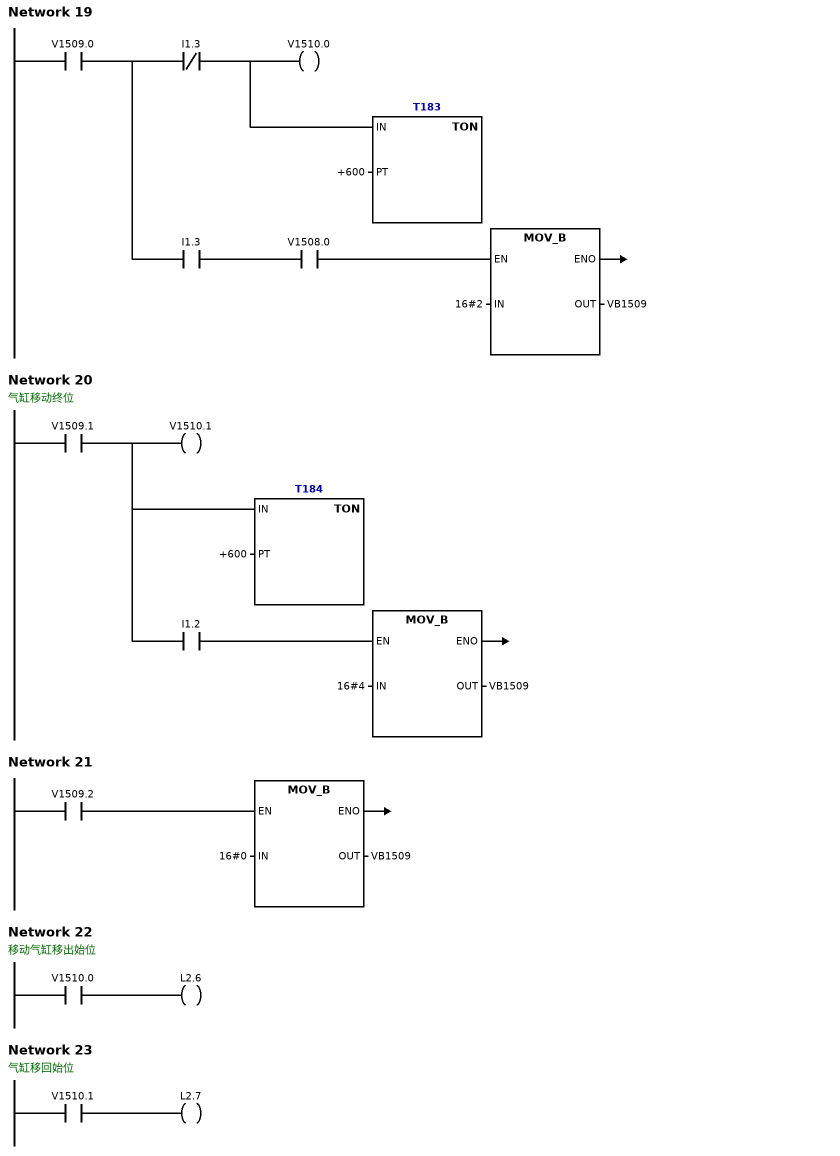
[picture p48: SBR10 networks 19-23]
Network 19
LD     V1509.0
LPS
AN     I1.3
=      V1510.0
TON    T183, +600
LPP
A      I1.3
A      V1508.0
MOVB   16#2, VB1509
Network 20
// 气缸移动终位
LD     V1509.1
=      V1510.1
TON    T184, +600
A      I1.2
MOVB   16#4, VB1509
Network 21
LD     V1509.2
MOVB   16#0, VB1509
Network 22
// 移动气缸移出始位
LD     V1510.0
=      L2.6
Network 23
// 气缸移回始位
LD     V1510.1
=      L2.7
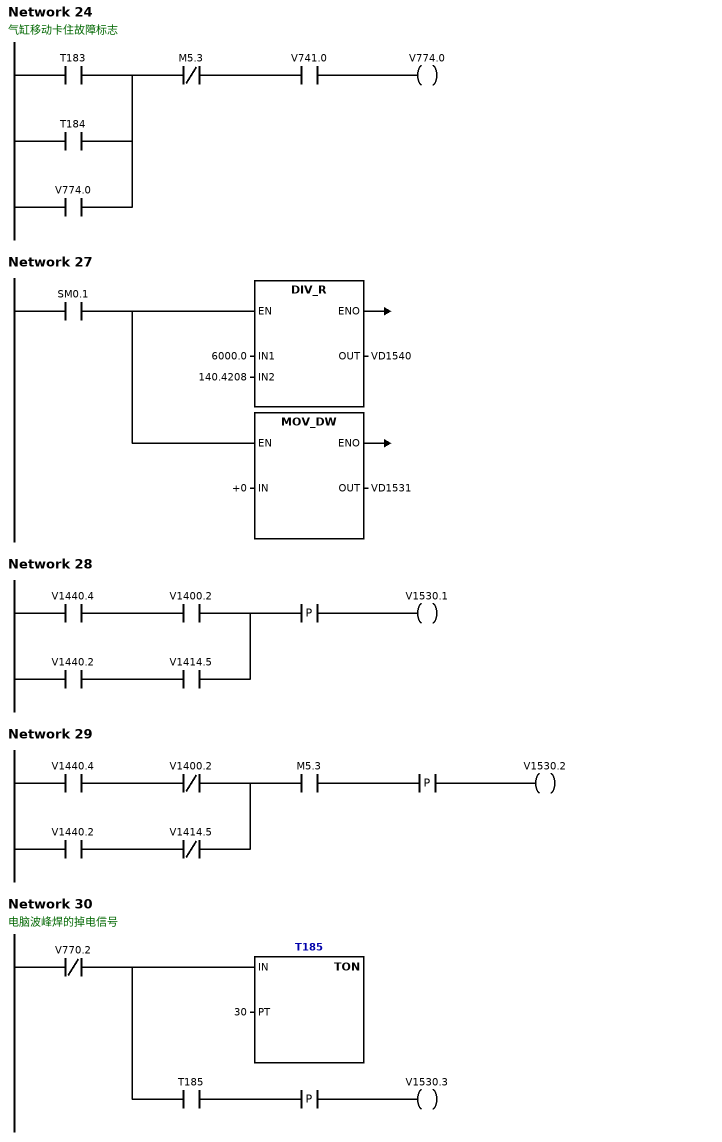
Network 24
// 气缸移动卡住故障标志
LD     T183
O      T184
O      V774.0
AN     M5.3
A      V741.0
=      V774.0
Network 27
LD     SM0.1
MOVR   6000.0, VD1540
/R     140.4208, VD1540
MOVD   +0, VD1531
Network 28
LD     V1440.4
A      V1400.2
LD     V1440.2
A      V1414.5
OLD
EU
=      V1530.1
Network 29
LD     V1440.4
AN     V1400.2
LD     V1440.2
AN     V1414.5
OLD
A      M5.3
EU
=      V1530.2
Network 30
// 电脑波峰焊的掉电信号
LDN    V770.2
TON    T185, 30
A      T185
EU
=      V1530.3
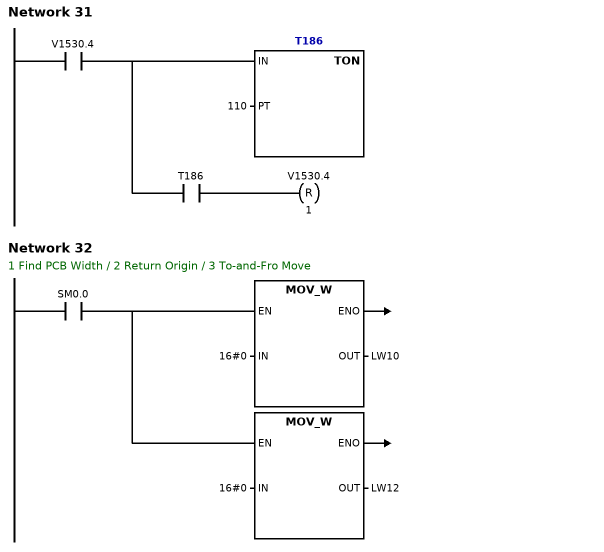
Network 31
LD     V1530.4
TON    T186, 110
A      T186
R      V1530.4, 1
Network 32
// 1 Find PCB Width
// 2 Return Origin
// 3 To-and-Fro Move
LD     SM0.0
MOVW   16#0, LW10
MOVW   16#0, LW12
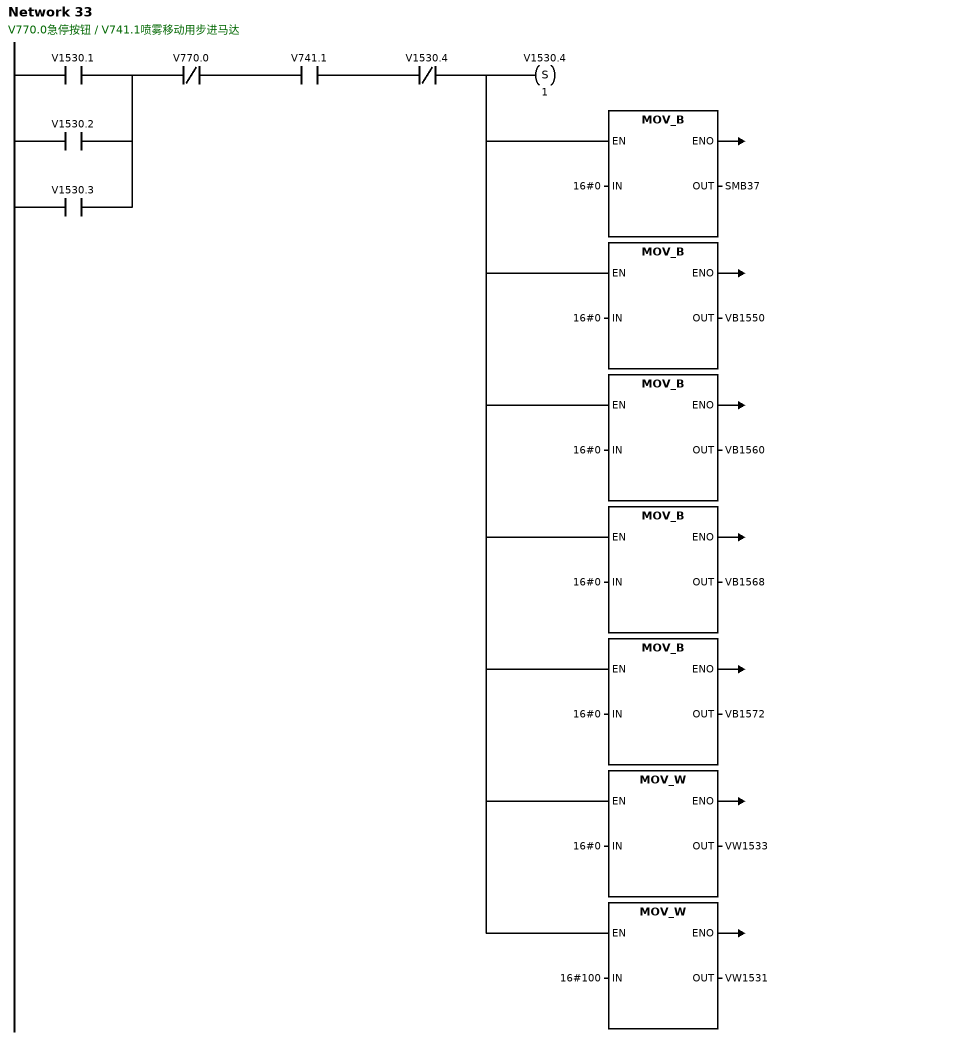
Network 33
// V770.0急停按钮
// V741.1喷雾移动用步进马达
LD     V1530.1
O      V1530.2
O      V1530.3
AN     V770.0
A      V741.1
AN     V1530.4
S      V1530.4, 1
MOVB   16#0, SMB37
MOVB   16#0, VB1550
MOVB   16#0, VB1560
MOVB   16#0, VB1568
MOVB   16#0, VB1572
MOVW   16#0, VW1533
MOVW   16#100, VW1531
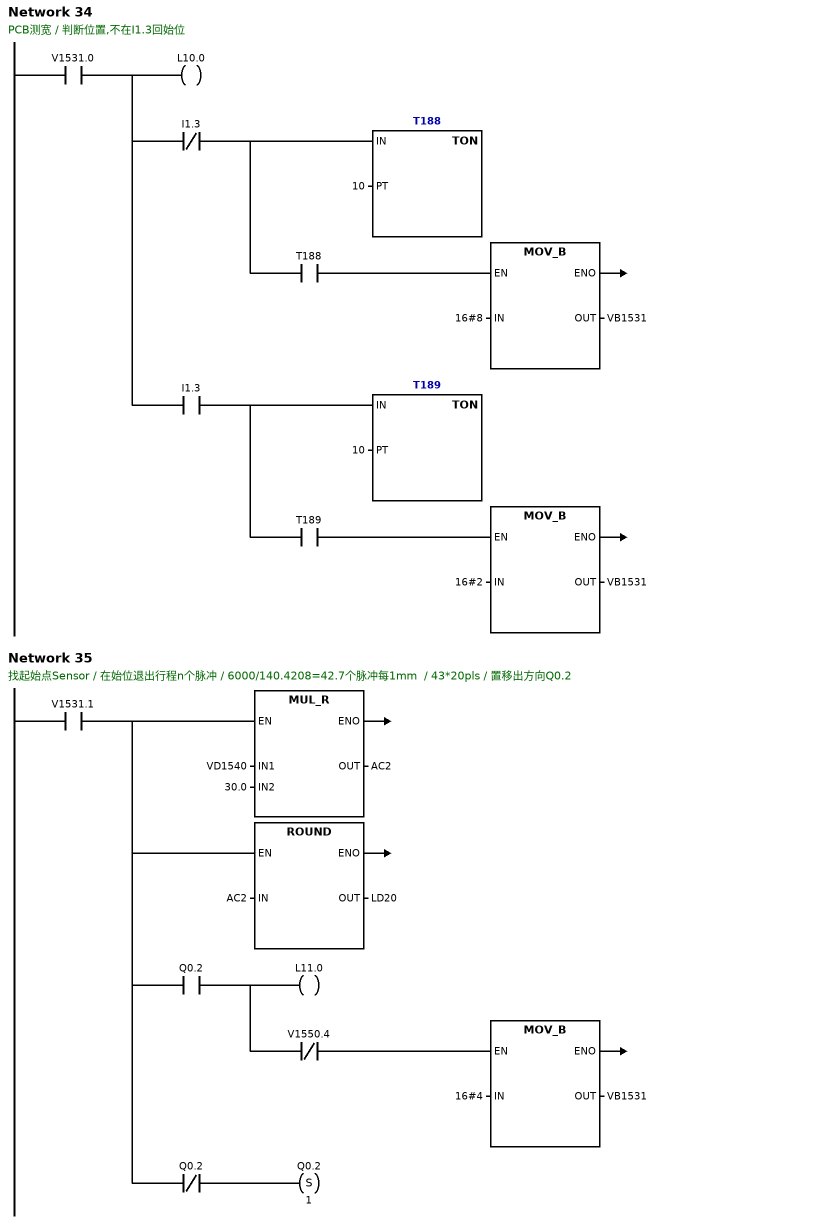
Network 34
// PCB测宽
// 判断位置,不在I1.3回始位
LD     V1531.0
LPS
=      L10.0
AN     I1.3
TON    T188, 10
A      T188
MOVB   16#8, VB1531
LPP
A      I1.3
TON    T189, 10
A      T189
MOVB   16#2, VB1531
Network 35
// 找起始点Sensor
// 在始位退出行程n个脉冲
// 6000/140.4208=42.7个脉冲每1mm 
// 43*20pls
// 置移出方向Q0.2
LD     V1531.1
LPS
MOVR   VD1540, AC2
*R     30.0, AC2
ROUND  AC2, LD20
A      Q0.2
=      L11.0
AN     V1550.4
MOVB   16#4, VB1531
LPP
AN     Q0.2
S      Q0.2, 1
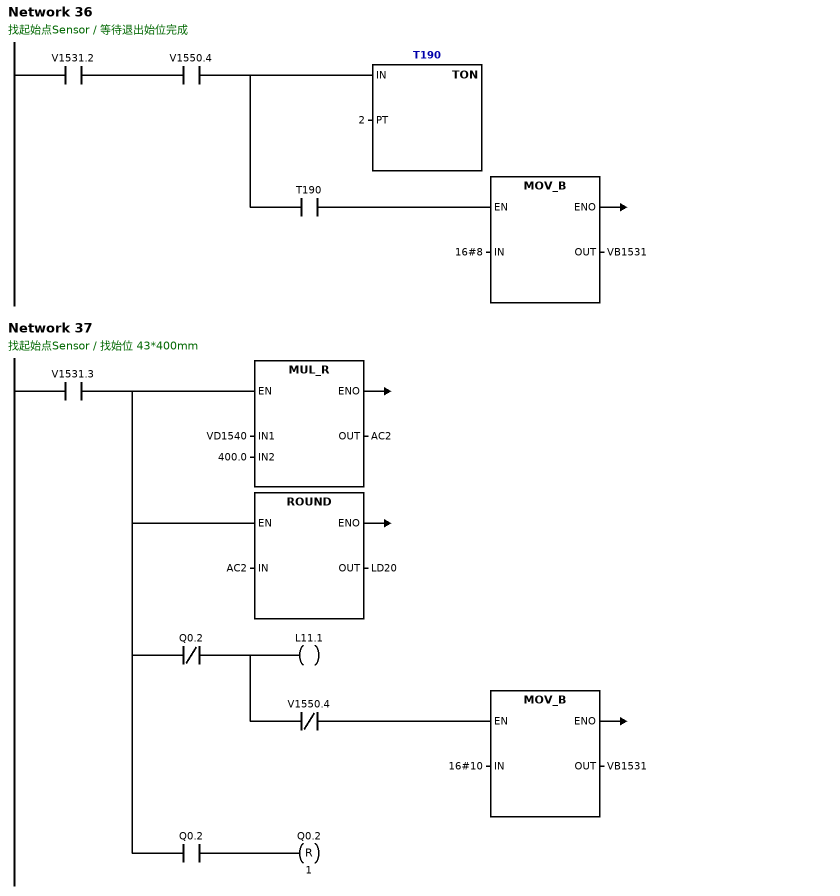
Network 36
// 找起始点Sensor
// 等待退出始位完成
LD     V1531.2
A      V1550.4
TON    T190, 2
A      T190
MOVB   16#8, VB1531
Network 37
// 找起始点Sensor
// 找始位 43*400mm
LD     V1531.3
LPS
MOVR   VD1540, AC2
*R     400.0, AC2
ROUND  AC2, LD20
AN     Q0.2
=      L11.1
AN     V1550.4
MOVB   16#10, VB1531
LPP
A      Q0.2
R      Q0.2, 1
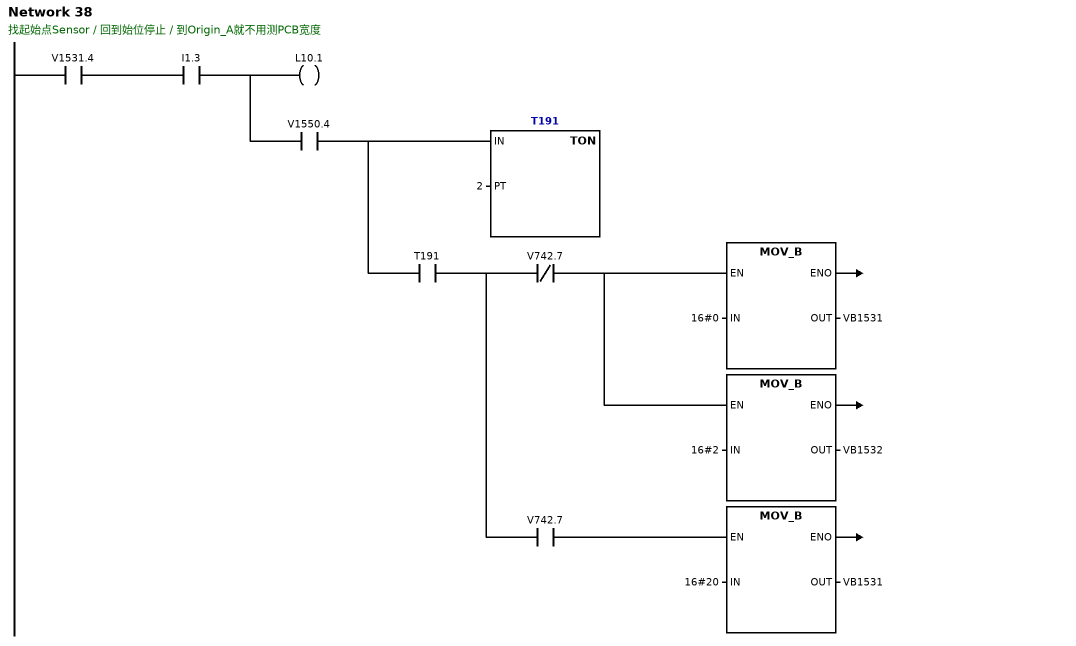
Network 38
// 找起始点Sensor
// 回到始位停止
// 到Origin_A就不用测PCB宽度
LD     V1531.4
A      I1.3
=      L10.1
A      V1550.4
TON    T191, 2
A      T191
LPS
AN     V742.7
MOVB   16#0, VB1531
MOVB   16#2, VB1532
LPP
A      V742.7
MOVB   16#20, VB1531
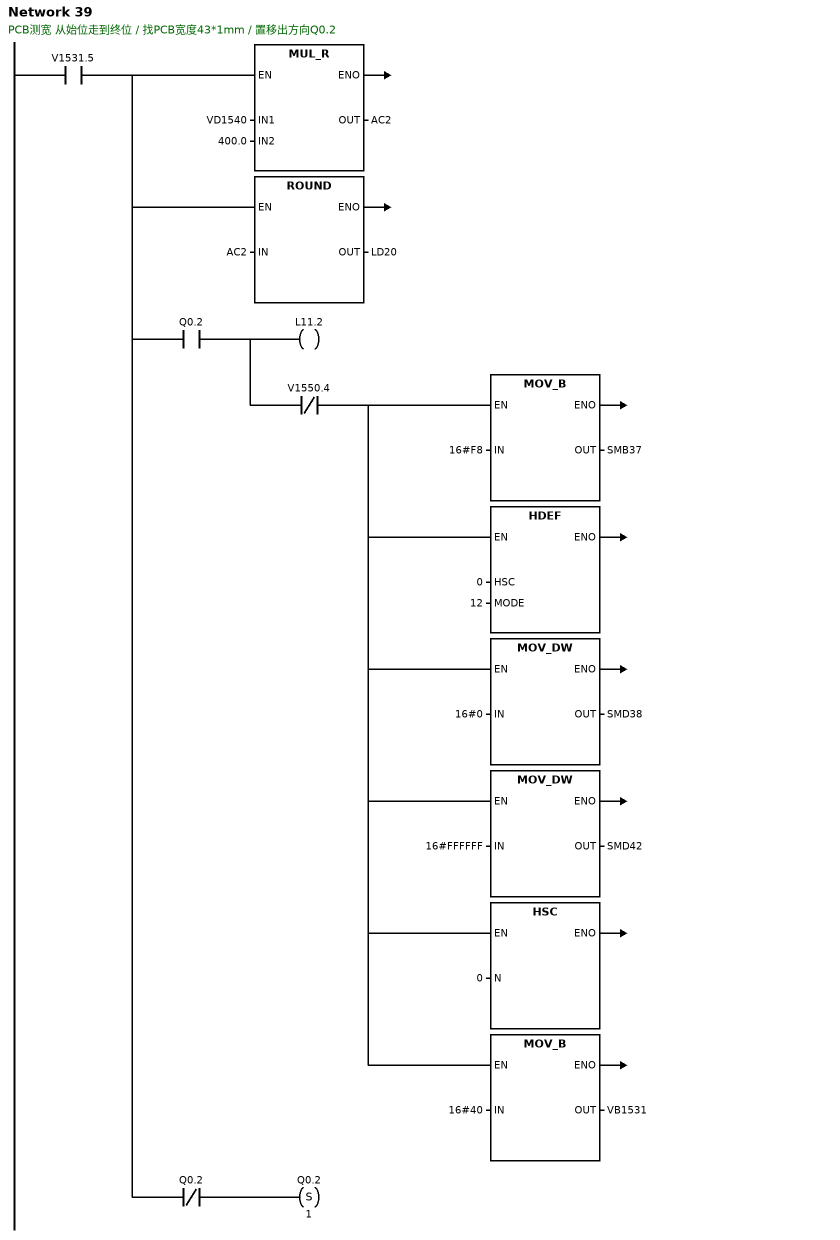
Network 39
// PCB测宽 从始位走到终位
// 找PCB宽度43*1mm
// 置移出方向Q0.2
LD     V1531.5
LPS
MOVR   VD1540, AC2
*R     400.0, AC2
ROUND  AC2, LD20
A      Q0.2
=      L11.2
AN     V1550.4
MOVB   16#F8, SMB37
HDEF   0, 12
MOVD   16#0, SMD38
MOVD   16#FFFFFF, SMD42
HSC    0
MOVB   16#40, VB1531
LPP
AN     Q0.2
S      Q0.2, 1
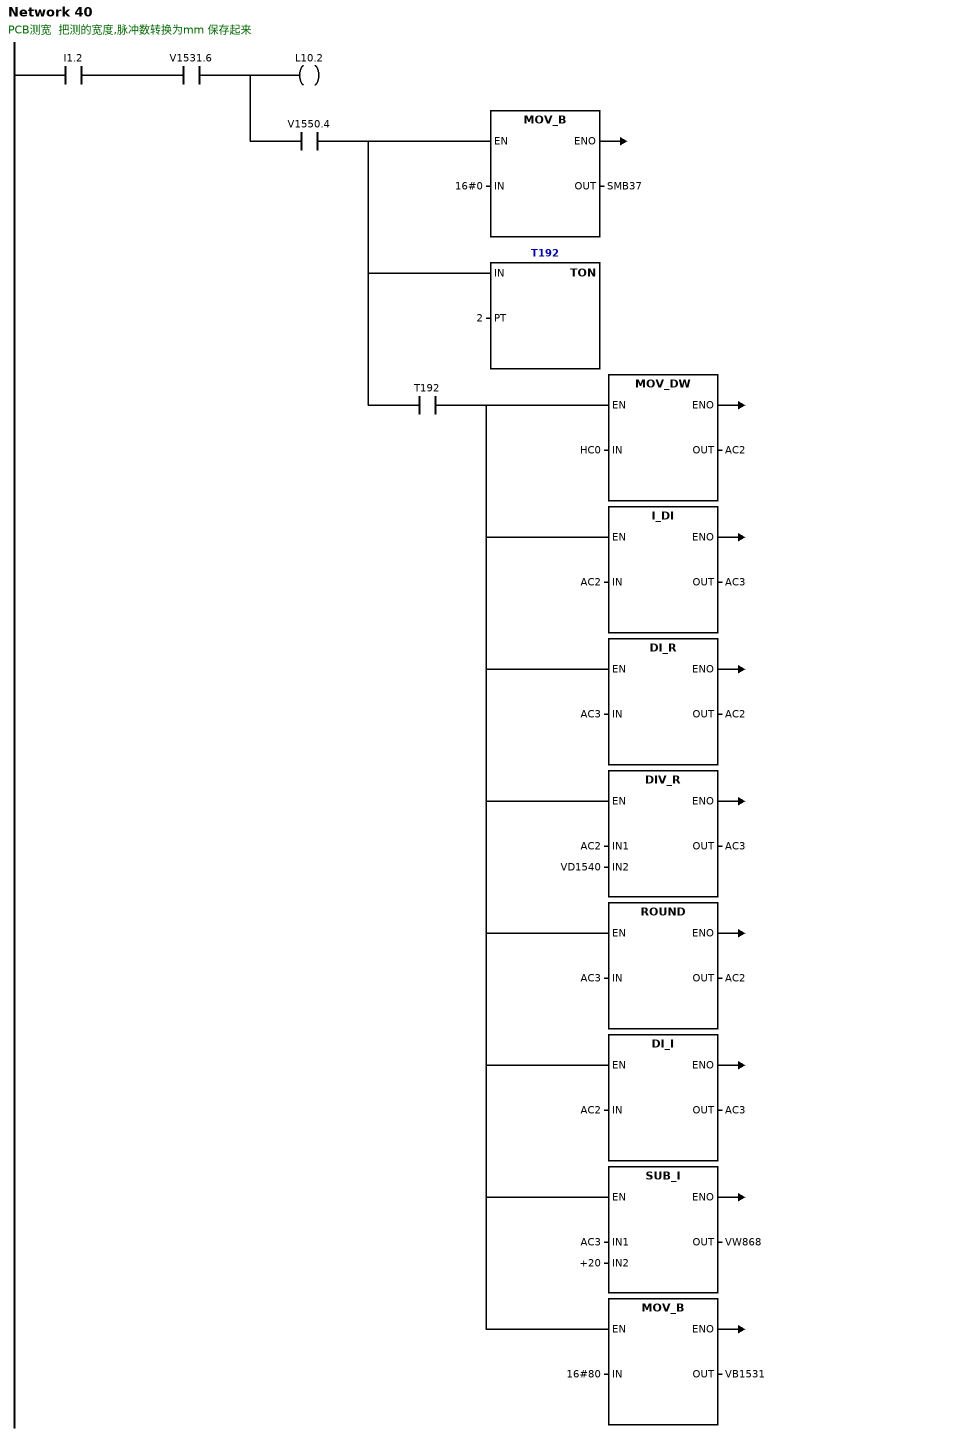
Network 40
// PCB测宽  把测的宽度,脉冲数转换为mm 保存起来
LD     I1.2
A      V1531.6
=      L10.2
A      V1550.4
MOVB   16#0, SMB37
TON    T192, 2
A      T192
MOVD   HC0, AC2
ITD    AC2, AC3
DTR    AC3, AC2
MOVR   AC2, AC3
/R     VD1540, AC3
ROUND  AC3, AC2
DTI    AC2, AC3
MOVW   AC3, VW868
-I     +20, VW868
MOVB   16#80, VB1531
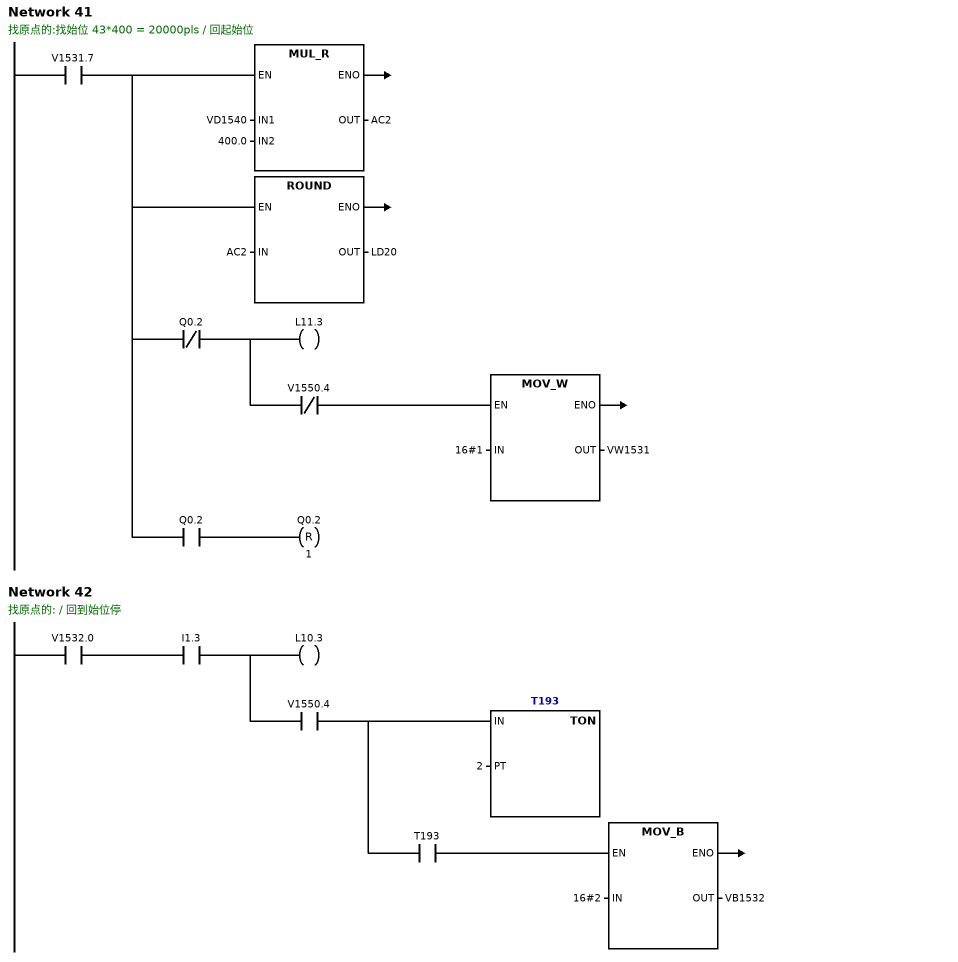
Network 41
// 找原点的:找始位 43*400 = 20000pls
// 回起始位
LD     V1531.7
LPS
MOVR   VD1540, AC2
*R     400.0, AC2
ROUND  AC2, LD20
AN     Q0.2
=      L11.3
AN     V1550.4
MOVW   16#1, VW1531
LPP
A      Q0.2
R      Q0.2, 1
Network 42
// 找原点的:
// 回到始位停
LD     V1532.0
A      I1.3
=      L10.3
A      V1550.4
TON    T193, 2
A      T193
MOVB   16#2, VB1532
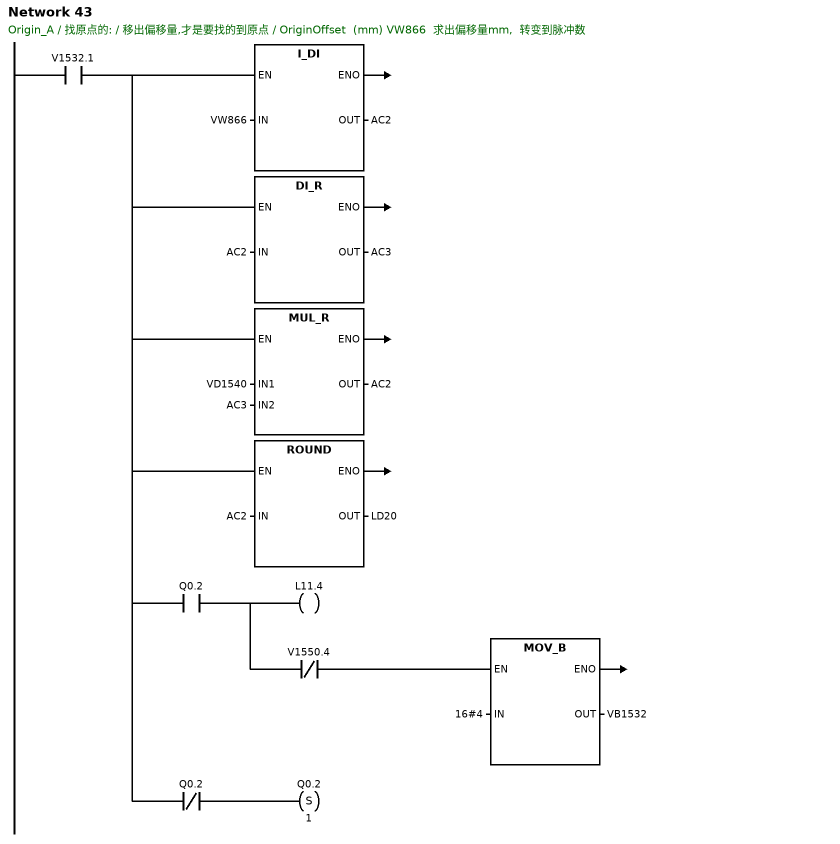
Network 43
// Origin_A
// 找原点的:
// 移出偏移量,才是要找的到原点
// OriginOffset  (mm) VW866  求出偏移量mm,  转变到脉冲数
LD     V1532.1
LPS
ITD    VW866, AC2
DTR    AC2, AC3
MOVR   VD1540, AC2
*R     AC3, AC2
ROUND  AC2, LD20
A      Q0.2
=      L11.4
AN     V1550.4
MOVB   16#4, VB1532
LPP
AN     Q0.2
S      Q0.2, 1
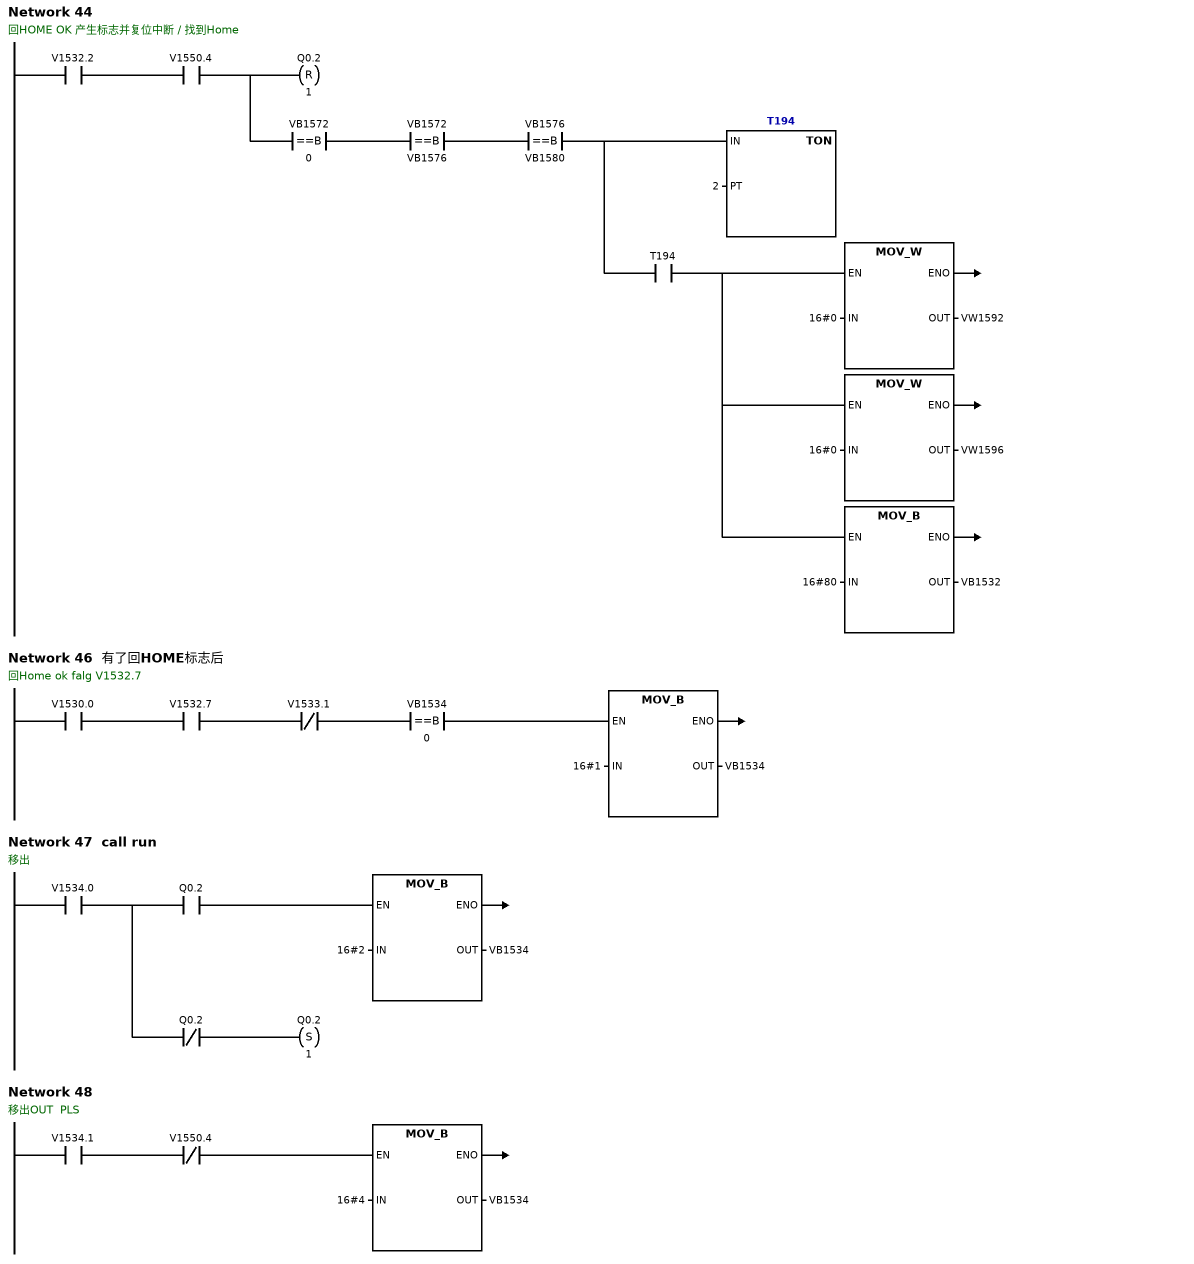
Network 44
// 回HOME OK 产生标志并复位中断
// 找到Home
LD     V1532.2
A      V1550.4
R      Q0.2, 1
AB=    VB1572, 0
AB=    VB1572, VB1576
AB=    VB1576, VB1580
TON    T194, 2
A      T194
MOVW   16#0, VW1592
MOVW   16#0, VW1596
MOVB   16#80, VB1532
Network 46 // 有了回HOME标志后
// 回Home ok falg V1532.7
LD     V1530.0
A      V1532.7
AN     V1533.1
AB=    VB1534, 0
MOVB   16#1, VB1534
Network 47 // call run
// 移出
LD     V1534.0
LPS
A      Q0.2
MOVB   16#2, VB1534
LPP
AN     Q0.2
S      Q0.2, 1
Network 48
// 移出OUT  PLS
LD     V1534.1
AN     V1550.4
MOVB   16#4, VB1534
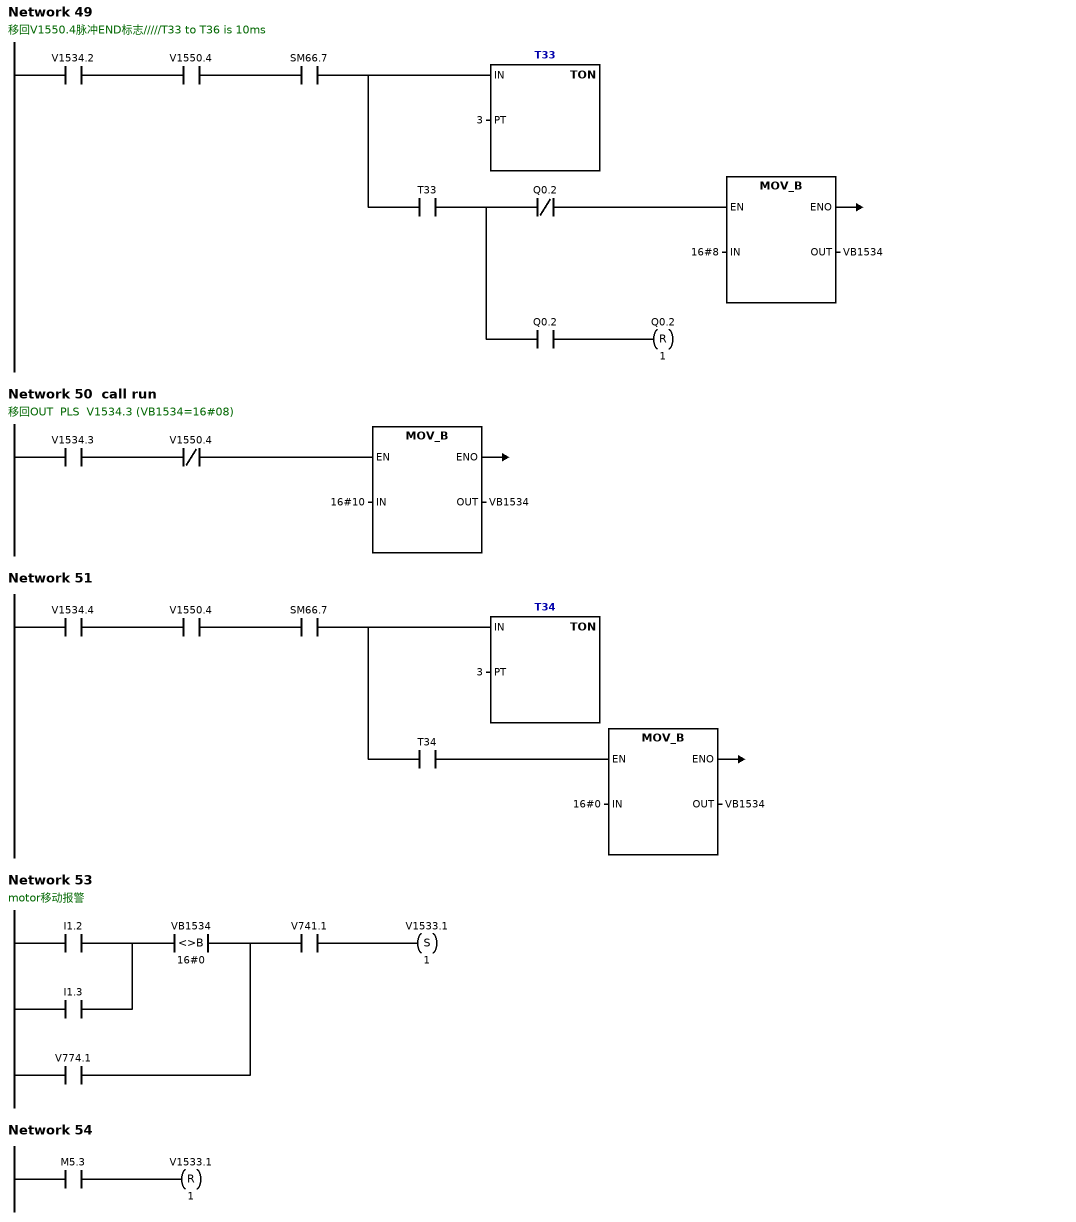
Network 49
// 移回V1550.4脉冲END标志/////T33 to T36 is 10ms
LD     V1534.2
A      V1550.4
A      SM66.7
TON    T33, 3
A      T33
LPS
AN     Q0.2
MOVB   16#8, VB1534
LPP
A      Q0.2
R      Q0.2, 1
Network 50 // call run
// 移回OUT  PLS  V1534.3 (VB1534=16#08)
LD     V1534.3
AN     V1550.4
MOVB   16#10, VB1534
Network 51
LD     V1534.4
A      V1550.4
A      SM66.7
TON    T34, 3
A      T34
MOVB   16#0, VB1534
Network 53
// motor移动报警
LD     I1.2
O      I1.3
AB<>   VB1534, 16#0
O      V774.1
A      V741.1
S      V1533.1, 1
Network 54
LD     M5.3
R      V1533.1, 1
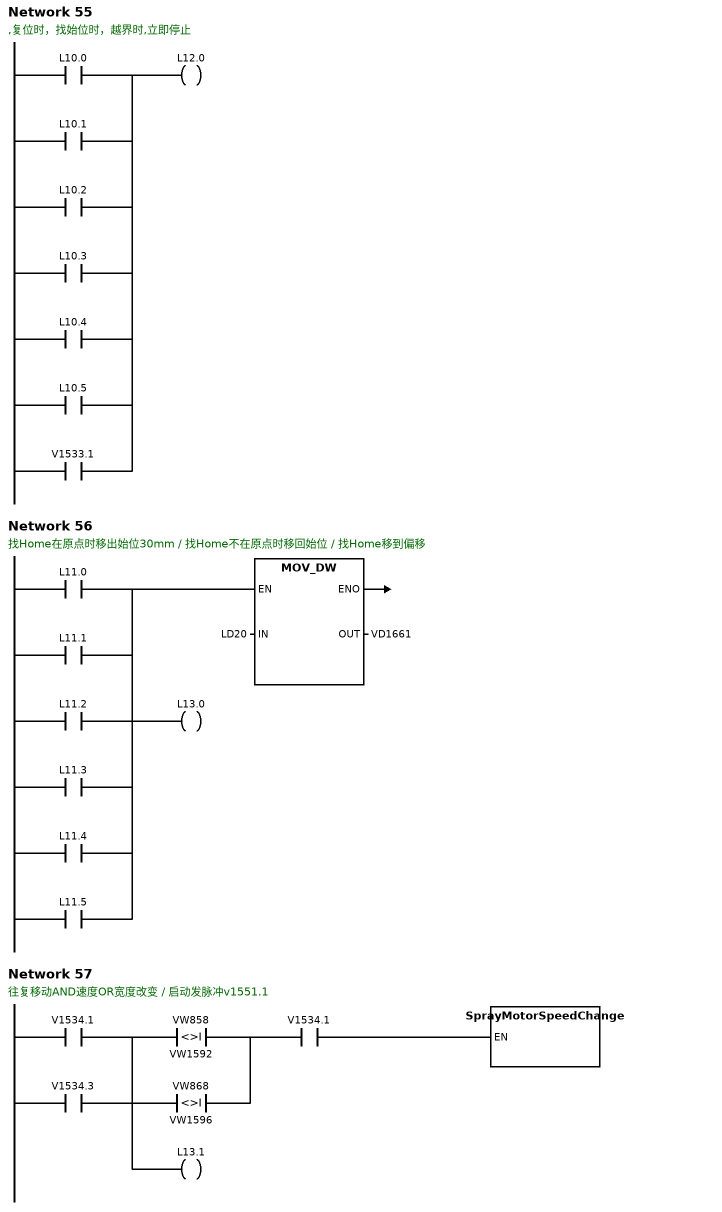
Network 55
// ,复位时，找始位时，越界时,立即停止
LD     L10.0
O      L10.1
O      L10.2
O      L10.3
O      L10.4
O      L10.5
O      V1533.1
=      L12.0
Network 56
// 找Home在原点时移出始位30mm
// 找Home不在原点时移回始位
// 找Home移到偏移
LD     L11.0
O      L11.1
O      L11.2
O      L11.3
O      L11.4
O      L11.5
MOVD   LD20, VD1661
=      L13.0
Network 57
// 往复移动AND速度OR宽度改变
// 启动发脉冲v1551.1
LD     V1534.1
O      V1534.3
LPS
LDW<>  VW858, VW1592
OW<>   VW868, VW1596
ALD
A      V1534.1
CALL   SprayMotorSpeedChange:SBR25
LPP
=      L13.1
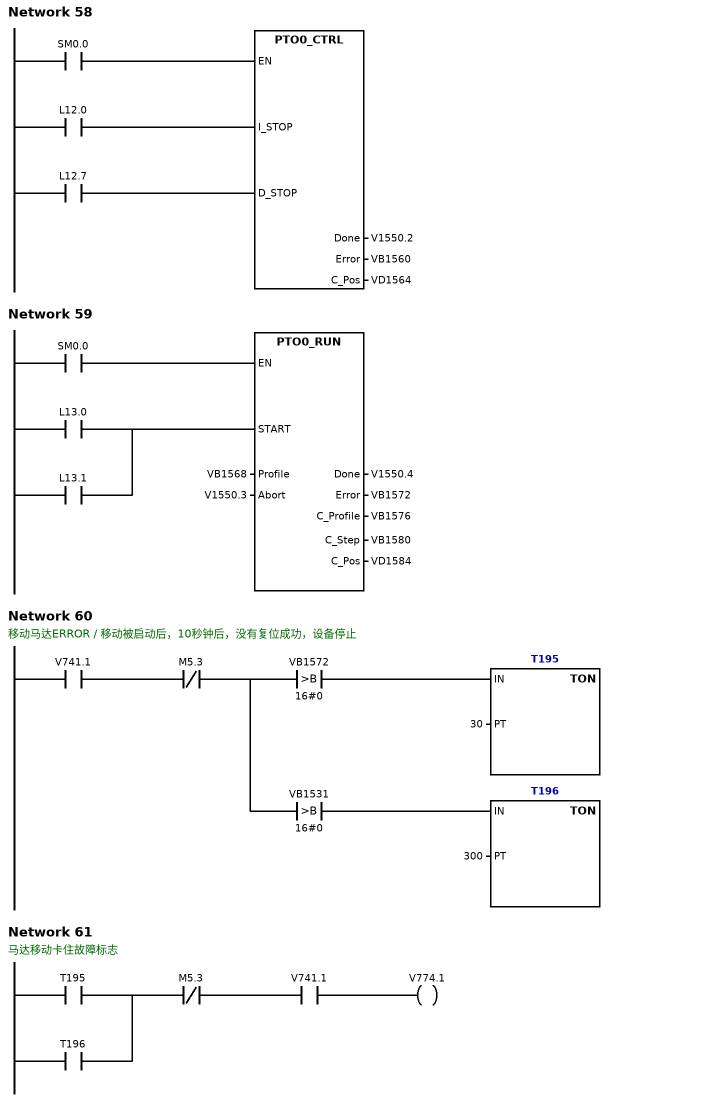
Network 58
LD     SM0.0
=      L60.0
LD     L12.0
=      L63.7
LD     L12.7
=      L63.6
LD     L60.0
CALL   PTO0_CTRL:SBR26, L63.7, L63.6, V1550.2, VB1560, VD1564
Network 59
LD     SM0.0
=      L60.0
LD     L13.0
O      L13.1
=      L63.7
LD     L60.0
CALL   PTO0_RUN:SBR27, L63.7, VB1568, V1550.3, V1550.4, VB1572, VB1576, VB1580, VD1584
Network 60
// 移动马达ERROR
// 移动被启动后，10秒钟后，没有复位成功，设备停止
LD     V741.1
AN     M5.3
LPS
AB>    VB1572, 16#0
TON    T195, 30
LPP
AB>    VB1531, 16#0
TON    T196, 300
Network 61
// 马达移动卡住故障标志
LD     T195
O      T196
AN     M5.3
A      V741.1
=      V774.1
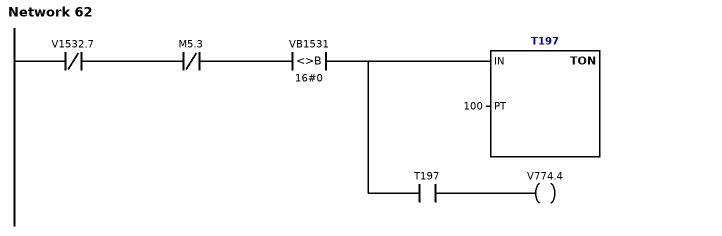
Network 62
LDN    V1532.7
AN     M5.3
AB<>   VB1531, 16#0
TON    T197, 100
A      T197
=      V774.4
END_SUBROUTINE_BLOCK

SUBROUTINE_BLOCK LiuLianDisVB2100_2199:SBR11
TITLE=Memory user VB2100  to  VB2199
BEGIN
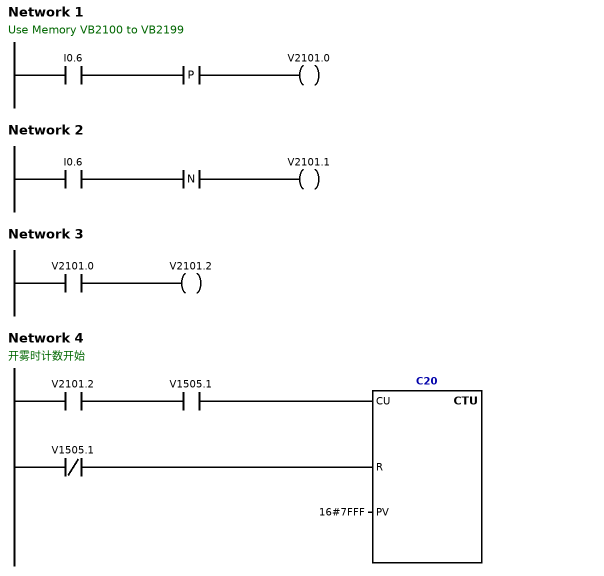
Network 1
// Use Memory VB2100 to VB2199
LD     I0.6
EU
=      V2101.0
Network 2
LD     I0.6
ED
=      V2101.1
Network 3
LD     V2101.0
=      V2101.2
Network 4
// 开雾时计数开始
LD     V2101.2
A      V1505.1
LDN    V1505.1
CTU    C20, 16#7FFF
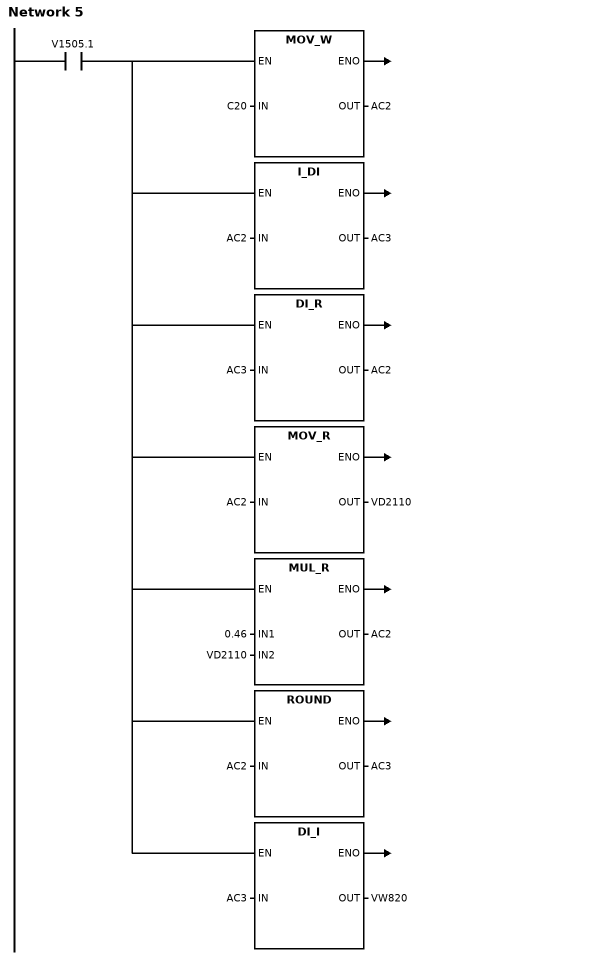
Network 5
LD     V1505.1
MOVW   C20, AC2
ITD    AC2, AC3
DTR    AC3, AC2
MOVR   AC2, VD2110
MOVR   0.46, AC2
*R     VD2110, AC2
ROUND  AC2, AC3
DTI    AC3, VW820
END_SUBROUTINE_BLOCK

SUBROUTINE_BLOCK ConveyWidthVB4000_4099:SBR16
TITLE=
BEGIN
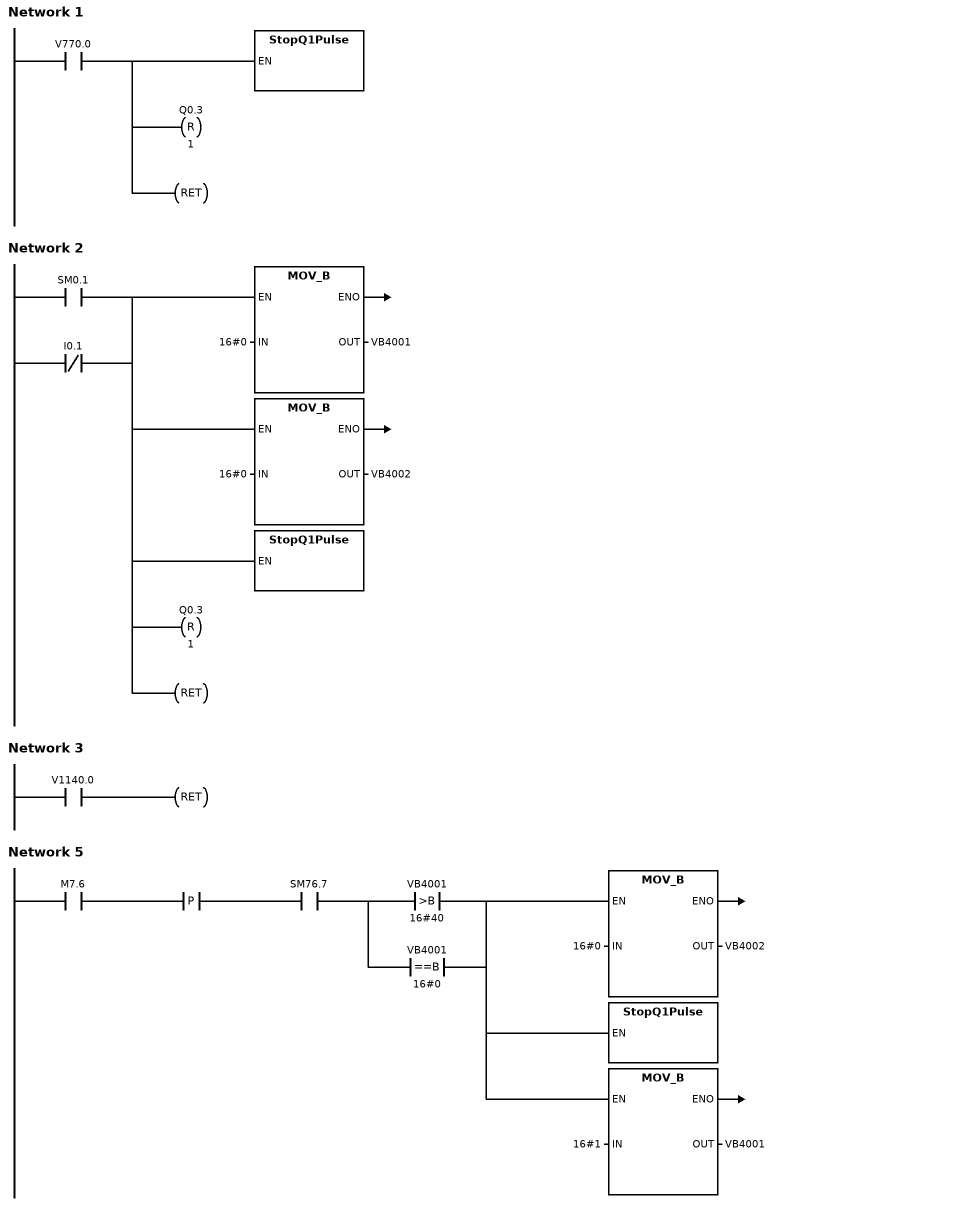
Network 1
LD     V770.0
CALL   StopQ1Pulse:SBR31
R      Q0.3, 1
CRET
Network 2
LD     SM0.1
ON     I0.1
MOVB   16#0, VB4001
MOVB   16#0, VB4002
CALL   StopQ1Pulse:SBR31
R      Q0.3, 1
CRET
Network 3
LD     V1140.0
CRET
Network 5
LD     M7.6
EU
A      SM76.7
LDB>   VB4001, 16#40
OB=    VB4001, 16#0
ALD
MOVB   16#0, VB4002
CALL   StopQ1Pulse:SBR31
MOVB   16#1, VB4001
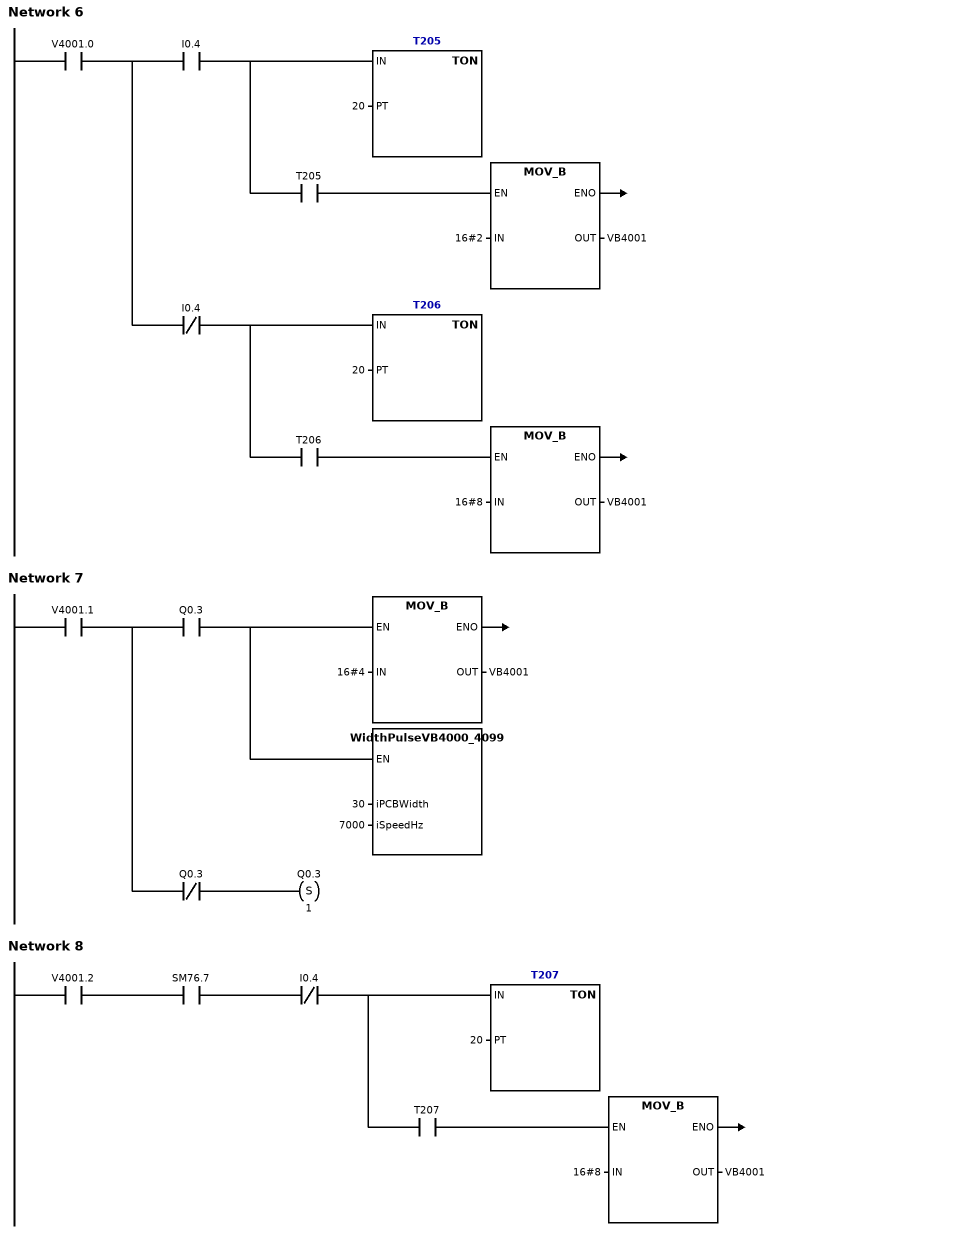
Network 6
LD     V4001.0
LPS
A      I0.4
TON    T205, 20
A      T205
MOVB   16#2, VB4001
LPP
AN     I0.4
TON    T206, 20
A      T206
MOVB   16#8, VB4001
Network 7
LD     V4001.1
LPS
A      Q0.3
MOVB   16#4, VB4001
CALL   WidthPulseVB4000_4099:SBR32, 30, 7000
LPP
AN     Q0.3
S      Q0.3, 1
Network 8
LD     V4001.2
A      SM76.7
AN     I0.4
TON    T207, 20
A      T207
MOVB   16#8, VB4001
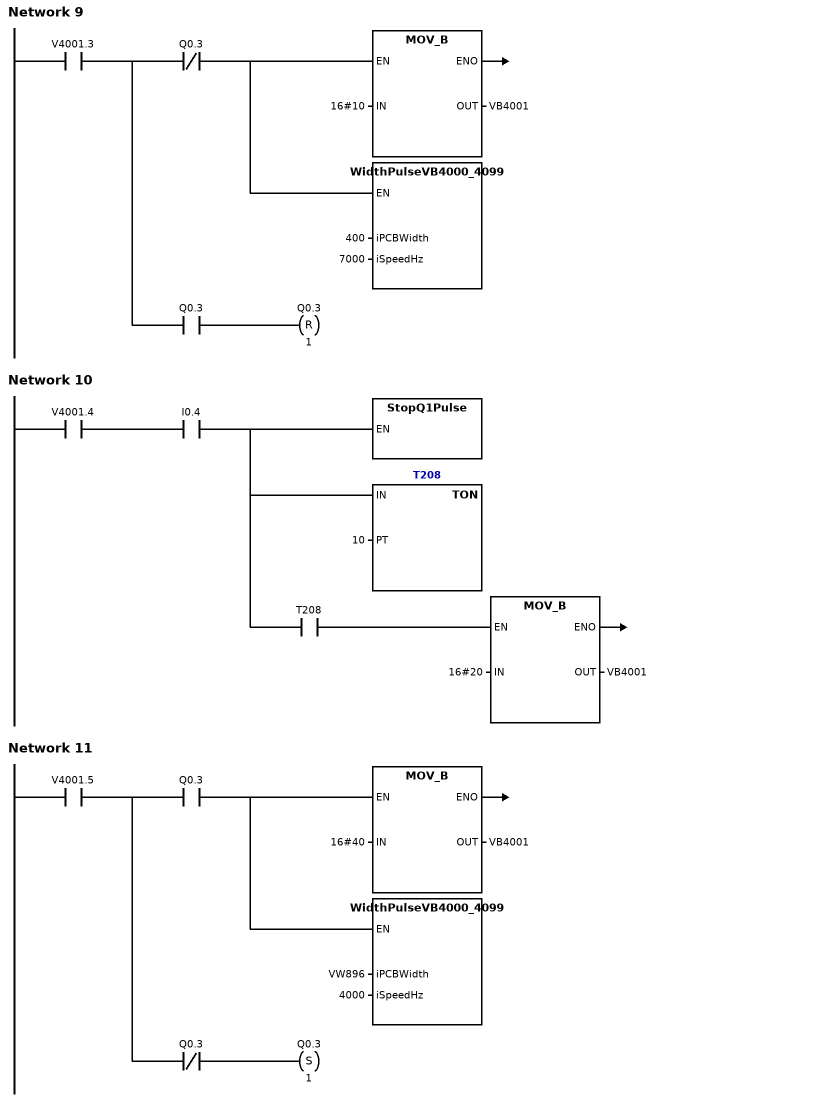
Network 9
LD     V4001.3
LPS
AN     Q0.3
MOVB   16#10, VB4001
CALL   WidthPulseVB4000_4099:SBR32, 400, 7000
LPP
A      Q0.3
R      Q0.3, 1
Network 10
LD     V4001.4
A      I0.4
CALL   StopQ1Pulse:SBR31
TON    T208, 10
A      T208
MOVB   16#20, VB4001
Network 11
LD     V4001.5
LPS
A      Q0.3
MOVB   16#40, VB4001
CALL   WidthPulseVB4000_4099:SBR32, VW896, 4000
LPP
AN     Q0.3
S      Q0.3, 1
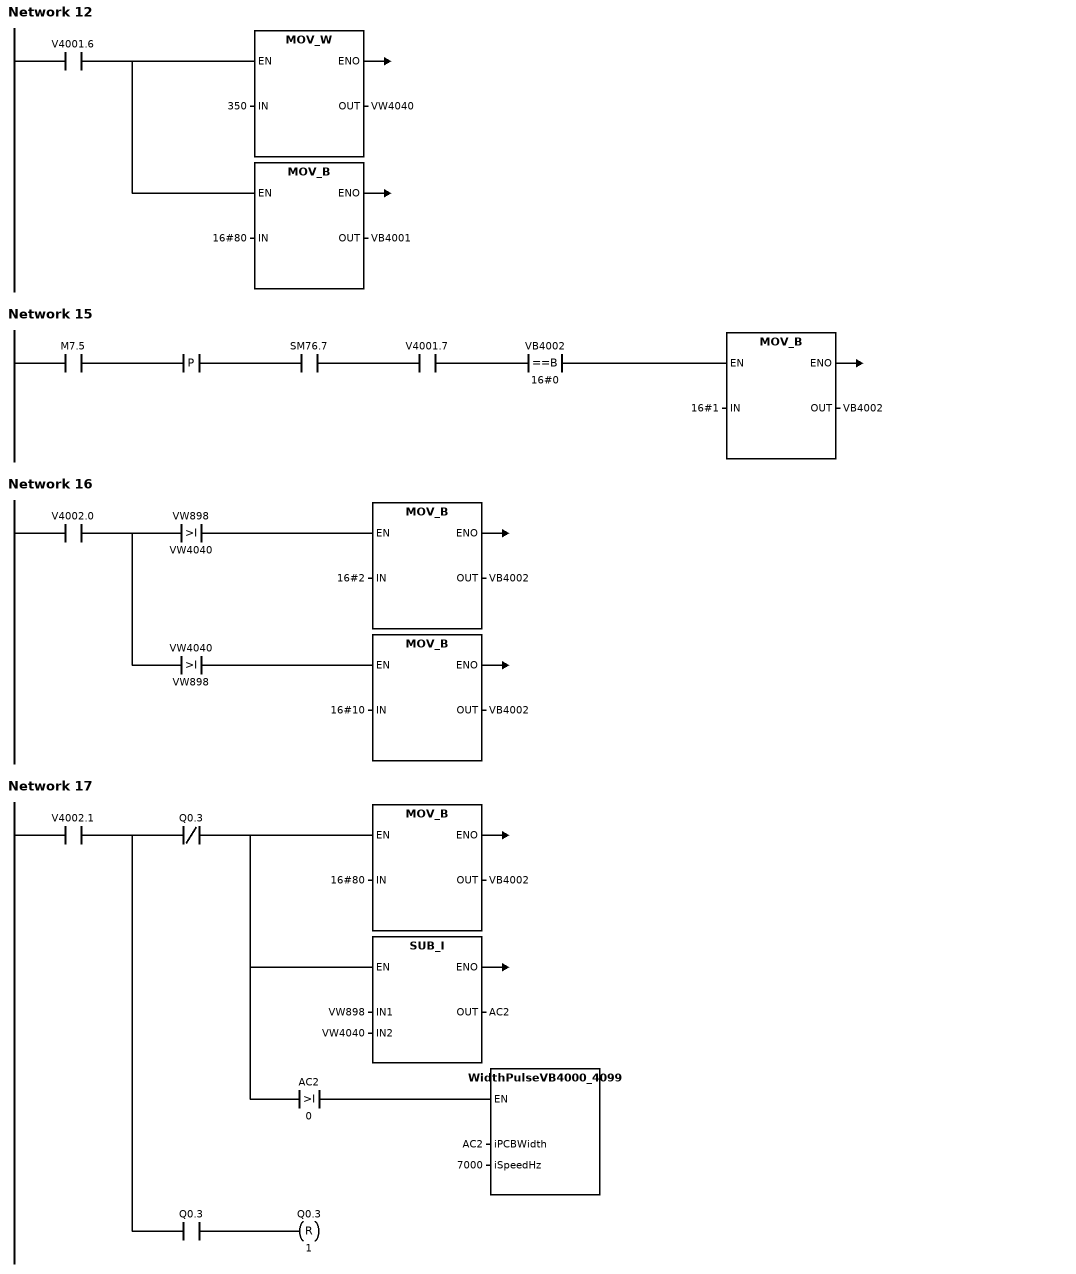
Network 12
LD     V4001.6
MOVW   350, VW4040
MOVB   16#80, VB4001
Network 15
LD     M7.5
EU
A      SM76.7
A      V4001.7
AB=    VB4002, 16#0
MOVB   16#1, VB4002
Network 16
LD     V4002.0
LPS
AW>    VW898, VW4040
MOVB   16#2, VB4002
LPP
AW>    VW4040, VW898
MOVB   16#10, VB4002
Network 17
LD     V4002.1
LPS
AN     Q0.3
MOVB   16#80, VB4002
MOVW   VW898, AC2
-I     VW4040, AC2
AW>    AC2, 0
CALL   WidthPulseVB4000_4099:SBR32, AC2, 7000
LPP
A      Q0.3
R      Q0.3, 1
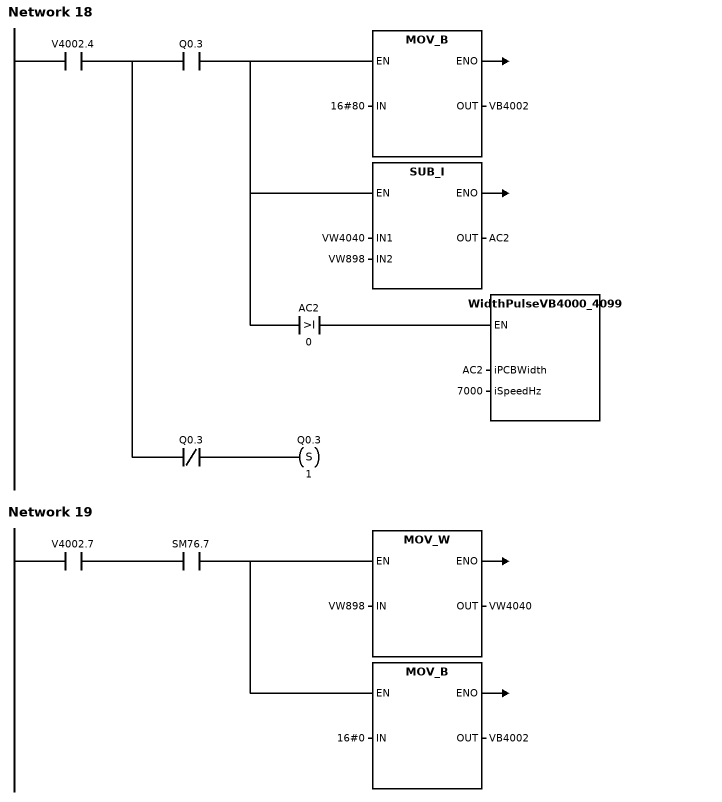
Network 18
LD     V4002.4
LPS
A      Q0.3
MOVB   16#80, VB4002
MOVW   VW4040, AC2
-I     VW898, AC2
AW>    AC2, 0
CALL   WidthPulseVB4000_4099:SBR32, AC2, 7000
LPP
AN     Q0.3
S      Q0.3, 1
Network 19
LD     V4002.7
A      SM76.7
MOVW   VW898, VW4040
MOVB   16#0, VB4002
END_SUBROUTINE_BLOCK

SUBROUTINE_BLOCK PCoperate3500_3999:SBR17
TITLE=
BEGIN
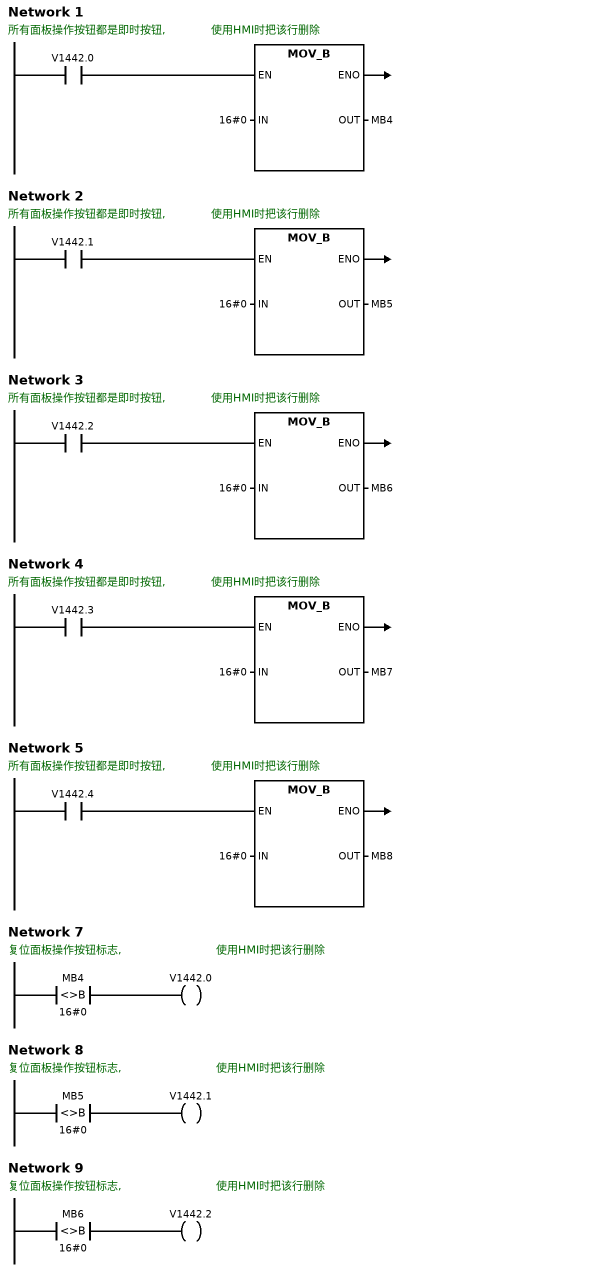
Network 1
// 所有面板操作按钮都是即时按钮,             使用HMI时把该行删除
LD     V1442.0
MOVB   16#0, MB4
Network 2
// 所有面板操作按钮都是即时按钮,             使用HMI时把该行删除
LD     V1442.1
MOVB   16#0, MB5
Network 3
// 所有面板操作按钮都是即时按钮,             使用HMI时把该行删除
LD     V1442.2
MOVB   16#0, MB6
Network 4
// 所有面板操作按钮都是即时按钮,             使用HMI时把该行删除
LD     V1442.3
MOVB   16#0, MB7
Network 5
// 所有面板操作按钮都是即时按钮,             使用HMI时把该行删除
LD     V1442.4
MOVB   16#0, MB8
Network 7
// 复位面板操作按钮标志,                           使用HMI时把该行删除
LDB<>  MB4, 16#0
=      V1442.0
Network 8
// 复位面板操作按钮标志,                           使用HMI时把该行删除
LDB<>  MB5, 16#0
=      V1442.1
Network 9
// 复位面板操作按钮标志,                           使用HMI时把该行删除
LDB<>  MB6, 16#0
=      V1442.2
